FUNCTION_BLOCK Trapizoidalf
VAR_INPUT
END_VAR
VAR_OUTPUT
END_VAR
VAR
END_VAR

END_FUNCTION_BLOCK

(* stored: Version 1.1.0.1, ProductVersion 3.1.4024.12
   POU Trapizoidalf: Id {e2e8732f-1814-4905-ac72-aa316cb52a81}, SpecialFunc None *)
